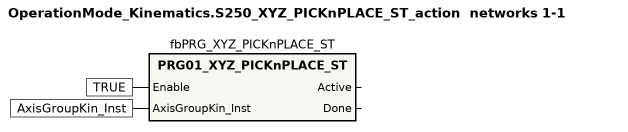
[picture p24: OperationMode_Kinematics.S250_XYZ_PICKnPLACE_ST_action (FBD) networks 1-1]
_FBD_ (* Function Block Diagram *)
NETWORK 1
	fbPRG_XYZ_PICKnPLACE_ST:PRG01_XYZ_PICKnPLACE_ST(Enable: TRUE, AxisGroupKin_Inst: AxisGroupKin_Inst)
_END_FBD_
(* the same logic as Structured Text *)
(* Network 1 *)
fbPRG_XYZ_PICKnPLACE_ST(Enable := TRUE, AxisGroupKin_Inst := AxisGroupKin_Inst);
END_ACTION

TRANSITION NOT referenced:
_FBD_ (* Function Block Diagram *)
NETWORK 1
	AND(AxisGroupKin_Inst.Out.General.Inverter.Connected[0], NOT AxisGroupKin_Inst.Out.General.Inverter.Referenced[0])
_END_FBD_
END_TRANSITION

TRANSITION referenced:
_FBD_ (* Function Block Diagram *)
NETWORK 1
	AND(AxisGroupKin_Inst.Out.General.Inverter.Connected[0], AxisGroupKin_Inst.Out.General.Inverter.Referenced[0])
_END_FBD_
END_TRANSITION

TRANSITION Homing done:
_FBD_ (* Function Block Diagram *)
NETWORK 1
	AND(AxisGroupKin_Inst.Out.General.Inverter.Connected[0], AxisGroupKin_Inst.Out.General.Inverter.Referenced[0])
_END_FBD_
END_TRANSITION

TRANSITION Automatic Mode:
_FBD_ (* Function Block Diagram *)
NETWORK 1
	AxisGroupKin_Inst.Out.General.Kin.Ready
_END_FBD_
(* the same logic as Structured Text *)
(* Network 1 *)
Automatic_Mode := AxisGroupKin_Inst.Out.General.Kin.Ready;
END_TRANSITION

TRANSITION Jog Mode:
_FBD_ (* Function Block Diagram *)
NETWORK 1
	NOT FALSE
_END_FBD_
(* the same logic as Structured Text *)
(* Network 1 *)
Jog_Mode := NOT FALSE;
END_TRANSITION

TRANSITION no Jog Mode:
_FBD_ (* Function Block Diagram *)
NETWORK 1
	FALSE
_END_FBD_
(* the same logic as Structured Text *)
(* Network 1 *)
no_Jog_Mode := FALSE;
END_TRANSITION

TRANSITION Start AND Enabled:
_FBD_ (* Function Block Diagram *)
NETWORK 1
	AND(TRUE, AxisGroupKin_Inst.Out.General.Kin.Ready)
_END_FBD_
END_TRANSITION

TRANSITION PRG1_Pick_and_Place_ST:
_FBD_ (* Function Block Diagram *)
NETWORK 1
	EQ(gKinExamples_Control[InstanceNumber].ProgramNumber, 1)
_END_FBD_
END_TRANSITION

TRANSITION Pick_and_Place_SFC:
_FBD_ (* Function Block Diagram *)
NETWORK 1
	EQ(gKinExamples_Control[InstanceNumber].ProgramNumber, 2)
_END_FBD_
END_TRANSITION

TRANSITION new Mode or Done:
_FBD_ (* Function Block Diagram *)
NETWORK 1
	OR(NE(gKinExamples_Control[InstanceNumber].ProgramNumber, 2), fbPRG_XYZ_PICKnPLACE_SFC.Done)
_END_FBD_
END_TRANSITION

TRANSITION XYZ_TARG_LIN_CIRC_ST:
_FBD_ (* Function Block Diagram *)
NETWORK 1
	EQ(gKinExamples_Control[InstanceNumber].ProgramNumber, 3)
_END_FBD_
END_TRANSITION

TRANSITION new Mode or Done:
_FBD_ (* Function Block Diagram *)
NETWORK 1
	OR(NE(gKinExamples_Control[InstanceNumber].ProgramNumber, 3), fbPRG_XYZ_TARG_LIN_CIRC_ST.Done)
_END_FBD_
END_TRANSITION

TRANSITION XYZ_TARG_LIN_CIRC_SFC:
_FBD_ (* Function Block Diagram *)
NETWORK 1
	EQ(gKinExamples_Control[InstanceNumber].ProgramNumber, 4)
_END_FBD_
END_TRANSITION

TRANSITION new Mode or Done:
_FBD_ (* Function Block Diagram *)
NETWORK 1
	OR(NE(gKinExamples_Control[InstanceNumber].ProgramNumber, 4), fbPRG_XYZ_TARG_LIN_CIRC_SFC.Done)
_END_FBD_
END_TRANSITION

TRANSITION XYZ_USER_ST:
_FBD_ (* Function Block Diagram *)
NETWORK 1
	EQ(gKinExamples_Control[InstanceNumber].ProgramNumber, 7)
_END_FBD_
END_TRANSITION

TRANSITION new Mode or Done:
_FBD_ (* Function Block Diagram *)
NETWORK 1
	OR(NE(gKinExamples_Control[InstanceNumber].ProgramNumber, 7), fbPRG_XYZ_USER_ST.Done)
_END_FBD_
END_TRANSITION

TRANSITION XYZ_USER_SFC:
_FBD_ (* Function Block Diagram *)
NETWORK 1
	EQ(gKinExamples_Control[InstanceNumber].ProgramNumber, 8)
_END_FBD_
END_TRANSITION

TRANSITION new Mode or Done:
_FBD_ (* Function Block Diagram *)
NETWORK 1
	OR(NE(gKinExamples_Control[InstanceNumber].ProgramNumber, 8), fbPRG_XYZ_USER_SFC.Done)
_END_FBD_
END_TRANSITION

TRANSITION FillQueue_LIN3D_with_Array_ST:
_FBD_ (* Function Block Diagram *)
NETWORK 1
	EQ(gKinExamples_Control[InstanceNumber].ProgramNumber, 5)
_END_FBD_
END_TRANSITION

TRANSITION new Mode or Done:
_FBD_ (* Function Block Diagram *)
NETWORK 1
	OR(NE(gKinExamples_Control[InstanceNumber].ProgramNumber, 5), fbPRG_XYZ_FillQueue_LIN3D_with_Array_ST.Done)
_END_FBD_
END_TRANSITION

TRANSITION FillQueue_LIN3D_with_Array_SFC:
_FBD_ (* Function Block Diagram *)
NETWORK 1
	EQ(gKinExamples_Control[InstanceNumber].ProgramNumber, 6)
_END_FBD_
END_TRANSITION

TRANSITION new Mode OR Done:
_FBD_ (* Function Block Diagram *)
NETWORK 1
	OR(NE(gKinExamples_Control[InstanceNumber].ProgramNumber, 6), fbPRG_XYZ_FillQueue_LIN3D_with_Array_SFC.Done)
_END_FBD_
END_TRANSITION

TRANSITION Jog Mode:
_FBD_ (* Function Block Diagram *)
NETWORK 1
	NOT FALSE
_END_FBD_
(* the same logic as Structured Text *)
(* Network 1 *)
Jog_Mode := NOT FALSE;
END_TRANSITION

TRANSITION new Mode or Done:
_FBD_ (* Function Block Diagram *)
NETWORK 1
	OR(NE(gKinExamples_Control[InstanceNumber].ProgramNumber, 1), fbPRG_XYZ_PICKnPLACE_ST.Done)
_END_FBD_
END_TRANSITION
END_FUNCTION_BLOCK

(* POU AxisGroupControl_Kinematics/Examples/PRG01_XYZ_PICKnPLACE_ST, ST *)
(*##############################################################################################################

	IMPORTANT NOTICE:
 	This example is a special and free service that demonstrates only the basic 
	approach to generating a PLC program as a non-binding sample. 
	SEW is not liable for the contents of the sample program.

	Name:			PRG_XYZ_PICKnPLACE_ST
	Job:			Example program		
					Sequence: XYZ_PICKnPLACE_P2 -> P3 -> P4 -> P3 -> P2 -> P1
					
################################################################################################################*)
FUNCTION_BLOCK  PRG01_XYZ_PICKnPLACE_ST
VAR_INPUT
	Enable : BOOL;
END_VAR
VAR_OUTPUT
	Active : BOOL;
	Done : BOOL;
END_VAR
VAR
	nState : INT := 0;
	fbRtrig : R_TRIG;
	i : INT;
END_VAR
VAR_IN_OUT
	AxisGroupKin_Inst											: ST_AxisGroupKin_Instance;
END_VAR
(* Initialisation at rising edge of VAR_INPUT Enable *)
fbRtrig(CLK:=Enable);
IF fbRtrig.Q THEN
	nState := 0;
	Active := TRUE;
END_IF

(* No execution, if Enable = False *)
IF (Enable = FALSE) THEN
	Done := FALSE;
	RETURN;
END_IF


CASE nState OF
0:	(*Start*)
	IF AxisGroupKin.ConfigDataAvailable THEN
		nState := 5;
	END_IF

5:	(* Up *)
	(* Initialize Kinematic Flags*)
	AxisGroupKin_Inst.In.Cp.Settings.PlusTargetCartABC:=FALSE;
	AxisGroupKin_Inst.In.Cp.Settings.UseMasterPosition:=FALSE;

(* TARGET_CART settings *)
	(* Motion Parameters *)
	AxisGroupKin_Inst.In.Target.Cart.Velocity := CART_VEL100;
	AxisGroupKin_Inst.In.Target.Cart.Acceleration := CART_ACC100;
	AxisGroupKin_Inst.In.Target.Cart.Deceleration := CART_DEC100;
	AxisGroupKin_Inst.In.Target.Cart.Jerk:=CART_Jerk100;
	AxisGroupKin_Inst.In.Target.Synchronization:= KIN_NO_SYNC;
	(* Coordinate System *)
	AxisGroupKin_Inst.In.Target.CoordSys:=KIN_KCS;

	AxisGroupKin_Inst.In.General.Mode := KIN_TARGET_CART;

	AxisGroupKin_Inst.In.Target.Position := XYZ_PICKnPLACE_P2;

	IF (MC_KinInProximity(Threshold := XYZ_PICKnPLACE_BlendingDistance,
			Position := AxisGroupKin_Inst.In.Target.Position,
			CoordSys := AxisGroupKin_Inst.In.Target.CoordSys,
			Dimension := 2#0000_0111, ActPos := AxisGroupKin_Inst.Out.General.Position)) THEN
		nState := 10;
	END_IF
	AxisGroupKin_Inst.In.Simu3D.Ctrl.Pen_TCP_WCS:=TRUE;

10:	(* Side *)
	AxisGroupKin_Inst.In.Target.Position := XYZ_PICKnPLACE_P3;
	IF (MC_KinInProximity(Threshold := XYZ_PICKnPLACE_BlendingDistance,
			Position := AxisGroupKin_Inst.In.Target.Position,
			CoordSys := AxisGroupKin_Inst.In.Target.CoordSys,
			Dimension := 2#0000_0111, ActPos := AxisGroupKin_Inst.Out.General.Position)) THEN
		nState := 20;
	END_IF

20:	(* Down *)
	AxisGroupKin_Inst.In.Target.Position := XYZ_PICKnPLACE_P4;
	IF (MC_KinInProximity(Threshold := 0.0,
			Position := AxisGroupKin_Inst.In.Target.Position,
			CoordSys := AxisGroupKin_Inst.In.Target.CoordSys,
			Dimension := 2#0000_0111, ActPos := AxisGroupKin_Inst.Out.General.Position)
			AND AxisGroupKin_Inst.Out.General.Standstill.ActCoordSys) THEN
		nState :=30;
	END_IF

30:	(* Up *)
	AxisGroupKin_Inst.In.Target.Position := XYZ_PICKnPLACE_P3;
	IF (MC_KinInProximity(Threshold := XYZ_PICKnPLACE_BlendingDistance,
			Position := AxisGroupKin_Inst.In.Target.Position,
			CoordSys := AxisGroupKin_Inst.In.Target.CoordSys,
			Dimension := 2#0000_0111, ActPos := AxisGroupKin_Inst.Out.General.Position)) THEN
		nState := 40;
	END_IF

40:	(* Side *)
	AxisGroupKin_Inst.In.Target.Position := XYZ_PICKnPLACE_P2;
	IF (MC_KinInProximity(Threshold := XYZ_PICKnPLACE_BlendingDistance,
			Position := AxisGroupKin_Inst.In.Target.Position,
			CoordSys := AxisGroupKin_Inst.In.Target.CoordSys,
			Dimension := 2#0000_0111, ActPos := AxisGroupKin_Inst.Out.General.Position)) THEN
		nState := 50;
	END_IF

50:	(* Down *)
	AxisGroupKin_Inst.In.Target.Position := XYZ_PICKnPLACE_P1;
	IF (MC_KinInProximity(Threshold := 0.0,
			Position := AxisGroupKin_Inst.In.Target.Position,
			CoordSys := AxisGroupKin_Inst.In.Target.CoordSys,
			Dimension := 2#0000_0111, ActPos := AxisGroupKin_Inst.Out.General.Position)
			AND AxisGroupKin_Inst.Out.General.Standstill.ActCoordSys) THEN
		AxisGroupKin_Inst.In.Simu3D.Ctrl.Pen_TCP_WCS:=FALSE;
		Done := TRUE;
		Active := FALSE;
	END_IF

ELSE
;

END_CASE
END_FUNCTION_BLOCK

(* POU AxisGroupControl_Kinematics/Examples/PRG02_XYZ_PICKnPLACE_SFC, SFC *)
(*##############################################################################################################

	IMPORTANT NOTICE:
 	This example is a special and free service that demonstrates only the basic 
	approach to generating a PLC program as a non-binding sample. 
	SEW is not liable for the contents of the sample program.

	Name:			PRG_XYZ_PICKnPLACE_SFC
	Job:			Example program		
					Sequence: XYZ_PICKnPLACE_P2 -> P3 -> P4 -> P3 -> P2 -> P1	

################################################################################################################*)
FUNCTION_BLOCK PRG02_XYZ_PICKnPLACE_SFC
VAR_INPUT
	SFCReset:BOOL;
	(*SFCInit:BOOL;*)
	SFCPause:BOOL;

	SFCTipMode:BOOL;
	SFCTip:BOOL;
	SFCEnableLimit:BOOL;
	SFCQuitError:BOOL;
END_VAR
VAR_OUTPUT
	SFCTrans:BOOL;
	SFCError:BOOL;
	SFCErrorStep:STRING;
	SFCErrorPOU:STRING;
	SFCCurrentStep:STRING;
	Done:BOOL;
END_VAR
VAR

END_VAR
VAR_IN_OUT
	AxisGroupKin_Inst											: ST_AxisGroupKin_Instance;
END_VAR
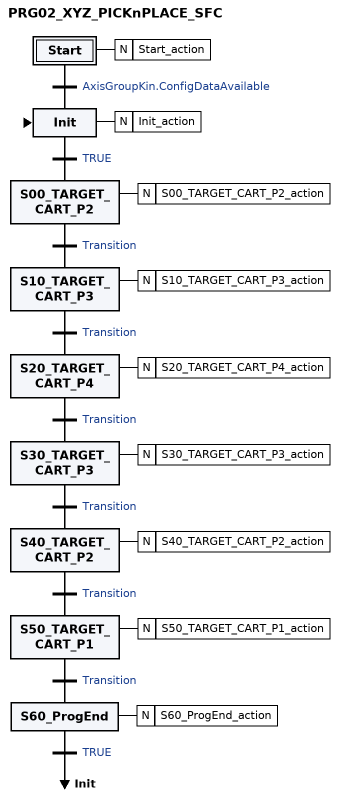
INITIAL_STEP Start:
	Start_action(N);
END_STEP
TRANSITION FROM Start TO Init := AxisGroupKin.ConfigDataAvailable;
END_TRANSITION
STEP Init:
	Init_action(N);
END_STEP
TRANSITION FROM Init TO S00_TARGET_CART_P2 := TRUE;
END_TRANSITION
STEP S00_TARGET_CART_P2:
	S00_TARGET_CART_P2_action(N);
END_STEP
TRANSITION FROM S00_TARGET_CART_P2 TO S10_TARGET_CART_P3 := Transition;
END_TRANSITION
STEP S10_TARGET_CART_P3:
	S10_TARGET_CART_P3_action(N);
END_STEP
TRANSITION FROM S10_TARGET_CART_P3 TO S20_TARGET_CART_P4 := Transition;
END_TRANSITION
STEP S20_TARGET_CART_P4:
	S20_TARGET_CART_P4_action(N);
END_STEP
TRANSITION FROM S20_TARGET_CART_P4 TO S30_TARGET_CART_P3 := Transition;
END_TRANSITION
STEP S30_TARGET_CART_P3:
	S30_TARGET_CART_P3_action(N);
END_STEP
TRANSITION FROM S30_TARGET_CART_P3 TO S40_TARGET_CART_P2 := Transition;
END_TRANSITION
STEP S40_TARGET_CART_P2:
	S40_TARGET_CART_P2_action(N);
END_STEP
TRANSITION FROM S40_TARGET_CART_P2 TO S50_TARGET_CART_P1 := Transition;
END_TRANSITION
STEP S50_TARGET_CART_P1:
	S50_TARGET_CART_P1_action(N);
END_STEP
TRANSITION FROM S50_TARGET_CART_P1 TO S60_ProgEnd := Transition;
END_TRANSITION
STEP S60_ProgEnd:
	S60_ProgEnd_action(N);
END_STEP
TRANSITION FROM S60_ProgEnd TO Init := TRUE;
END_TRANSITION

ACTION Start_action:
Done:=FALSE;
END_ACTION

ACTION Init_action:
(* Initialize Kinematic Flags*)
	AxisGroupKin_Inst.In.Cp.Settings.PlusTargetCartABC:=FALSE;
	AxisGroupKin_Inst.In.Cp.Settings.UseMasterPosition:=FALSE;

(* TARGET_CART settings *)
	(* Motion Parameters *)
	AxisGroupKin_Inst.In.Target.Cart.Velocity := CART_VEL100;
	AxisGroupKin_Inst.In.Target.Cart.Acceleration := CART_ACC100;
	AxisGroupKin_Inst.In.Target.Cart.Deceleration := CART_DEC100;
	AxisGroupKin_Inst.In.Target.Cart.Jerk := CART_Jerk100;
	AxisGroupKin_Inst.In.Target.Synchronization := KIN_NO_SYNC;
	(* Coordinate System *)
	AxisGroupKin_Inst.In.Target.CoordSys := KIN_KCS;

	AxisGroupKin_Inst.In.General.Mode := KIN_TARGET_CART;
END_ACTION

ACTION S00_TARGET_CART_P2_action:
AxisGroupKin_Inst.In.Target.Position := XYZ_PICKnPLACE_P2;
END_ACTION

ACTION S10_TARGET_CART_P3_action:
AxisGroupKin_Inst.In.Target.Position := XYZ_PICKnPLACE_P3;
END_ACTION

ACTION S20_TARGET_CART_P4_action:
AxisGroupKin_Inst.In.Target.Position := XYZ_PICKnPLACE_P4;
END_ACTION

ACTION S30_TARGET_CART_P3_action:
AxisGroupKin_Inst.In.Target.Position := XYZ_PICKnPLACE_P3;
END_ACTION

ACTION S40_TARGET_CART_P2_action:
AxisGroupKin_Inst.In.Target.Position := XYZ_PICKnPLACE_P2;
END_ACTION

ACTION S50_TARGET_CART_P1_action:
AxisGroupKin_Inst.In.Target.Position := XYZ_PICKnPLACE_P1;
END_ACTION

ACTION S60_ProgEnd_action:
Done:=TRUE;
END_ACTION

TRANSITION Transition:
MC_KinInProximity(Threshold := XYZ_PICKnPLACE_BlendingDistance,
			Position := AxisGroupKin_Inst.In.Target.Position,
			CoordSys := AxisGroupKin_Inst.In.Target.CoordSys,
			Dimension := 2#0000_0111, ActPos := AxisGroupKin_Inst.Out.General.Position)
END_TRANSITION

TRANSITION Transition:
MC_KinInProximity(Threshold := XYZ_PICKnPLACE_BlendingDistance,
			Position := AxisGroupKin_Inst.In.Target.Position,
			CoordSys := AxisGroupKin_Inst.In.Target.CoordSys,
			Dimension := 2#0000_0111, ActPos := AxisGroupKin_Inst.Out.General.Position)
END_TRANSITION

TRANSITION Transition:
MC_KinInProximity(Threshold := 0.0,
			Position := AxisGroupKin_Inst.In.Target.Position,
			CoordSys := AxisGroupKin_Inst.In.Target.CoordSys,
			Dimension := 2#0000_0111, ActPos := AxisGroupKin_Inst.Out.General.Position)
AND
AxisGroupKin_Inst.Out.General.Standstill.ActCoordSys
END_TRANSITION

TRANSITION Transition:
MC_KinInProximity(Threshold := XYZ_PICKnPLACE_BlendingDistance,
			Position := AxisGroupKin_Inst.In.Target.Position,
			CoordSys := AxisGroupKin_Inst.In.Target.CoordSys,
			Dimension := 2#0000_0111, ActPos := AxisGroupKin_Inst.Out.General.Position)
END_TRANSITION

TRANSITION Transition:
MC_KinInProximity(Threshold := XYZ_PICKnPLACE_BlendingDistance,
			Position := AxisGroupKin_Inst.In.Target.Position,
			CoordSys := AxisGroupKin_Inst.In.Target.CoordSys,
			Dimension := 2#0000_0111, ActPos := AxisGroupKin_Inst.Out.General.Position)
END_TRANSITION

TRANSITION Transition:
MC_KinInProximity(Threshold := 0.0,
			Position := AxisGroupKin_Inst.In.Target.Position,
			CoordSys := AxisGroupKin_Inst.In.Target.CoordSys,
			Dimension := 2#0000_0111, ActPos := AxisGroupKin_Inst.Out.General.Position)
AND
AxisGroupKin_Inst.Out.General.Standstill.ActCoordSys
END_TRANSITION
END_FUNCTION_BLOCK

(* POU AxisGroupControl_Kinematics/Examples/PRG03_XYZ_TARG_LIN_CIRC_ST, ST *)
(*##############################################################################################################

	IMPORTANT NOTICE:
 	This example is a special and free service that demonstrates only the basic 
	approach to generating a PLC program as a non-binding sample. 
	SEW is not liable for the contents of the sample program.

	Name:			PRG_XYZ_TARG_LIN_CIRC_ST
	Job:			Example program			
					Sequence: TARGET_CART to XYZ_TARG_LIN_CIRC_P1 -> LIN_XY to P2 -> CIRC_XZ with R3/A3 -> LIN_3D to P4 -> LIN_XY to P1

################################################################################################################*)
FUNCTION_BLOCK PRG03_XYZ_TARG_LIN_CIRC_ST
VAR_INPUT
	Enable : BOOL;
END_VAR
VAR_OUTPUT
	Active : BOOL;
	Done : BOOL;
END_VAR
VAR
	nState : INT;
	fbRtrig : R_TRIG;
END_VAR
VAR_IN_OUT
	AxisGroupKin_Inst											: ST_AxisGroupKin_Instance;
END_VAR
(* Initialisation at rising edge of VAR_INPUT Enable *)
fbRtrig(CLK:=Enable);
IF fbRtrig.Q THEN
	nState	:= 0;
	Active := TRUE;
END_IF

(* No execution, if Enable = False *)
IF NOT Enable THEN
	Done := FALSE;
	RETURN;
END_IF


CASE nState OF
0:	(*Start*)
	IF AxisGroupKin.ConfigDataAvailable THEN
		nState := 5;
	END_IF
5:	(* TARGET_CART to XYZ_TARG_LIN_CIRC_P1 *)
	(* Initialize Kinematic Flags*)
	AxisGroupKin_Inst.In.Cp.Settings.PlusTargetCartABC:=FALSE;
	AxisGroupKin_Inst.In.Cp.Settings.UseMasterPosition:=FALSE;

(* TARGET_CART settings *)
	(* Motion Parameters *)
	AxisGroupKin_Inst.In.Target.Cart.Acceleration := CART_ACC50;
	AxisGroupKin_Inst.In.Target.Cart.Deceleration := CART_DEC50;
	AxisGroupKin_Inst.In.Target.Cart.Velocity := CART_VEL50;
	AxisGroupKin_Inst.In.Target.Cart.Jerk:=CART_Jerk100;
	AxisGroupKin_Inst.In.Target.Synchronization:= KIN_NO_SYNC;
	(* Coordinate System *)
	AxisGroupKin_Inst.In.Target.CoordSys:=KIN_KCS;

	AxisGroupKin_Inst.In.General.Mode := KIN_TARGET_CART;

	AxisGroupKin_Inst.In.Target.Position := XYZ_TARG_LIN_CIRC_P1;
	IF (MC_KinInProximity(Threshold := 0.0,
			Position := AxisGroupKin_Inst.In.Target.Position,
			CoordSys := AxisGroupKin_Inst.In.Target.CoordSys,
			Dimension := 2#0000_0111, ActPos := AxisGroupKin_Inst.Out.General.Position)
			AND AxisGroupKin_Inst.Out.General.Standstill.ActCoordSys) THEN
		nState := 10;
	END_IF

10:	(* Straight line to XYZ_TARG_LIN_CIRC_P2, as soon as XYZ_TARG_LIN_CIRC_P1 has been reached *)

		AxisGroupKin_Inst.In.General.Mode := KIN_LIN_XY;
		AxisGroupKin_Inst.In.Cp.Segment.Position := XYZ_TARG_LIN_CIRC_P2;
(* CP motion parameters *)
		(* settings for whole path / all segments *)
		AxisGroupKin_Inst.In.Cp.Path.VelocityPercentage:=100;
		AxisGroupKin_Inst.In.Cp.Path.FidelityPercentage :=100;
		(* Settings for the segment, which should be added to the queue *)
		AxisGroupKin_Inst.In.Cp.Segment.Translation.Velocity := 1000;
		AxisGroupKin_Inst.In.Cp.Segment.Translation.Acceleration := 100;
		AxisGroupKin_Inst.In.Cp.Segment.Translation.Deceleration := 100;
		AxisGroupKin_Inst.In.Cp.Segment.Translation.Jerk := 100;
		AxisGroupKin_Inst.In.Cp.Segment.Blending.Distance := 50;
		AxisGroupKin_Inst.In.Cp.Segment.Blending.LimitationPercentage := 50;

		AxisGroupKin_Inst.In.Cp.Segment.ID := AxisGroupKin_Inst.In.Cp.Segment.ID + 1;	(* Change the SegmentID to add the segment to the queue *)

		AxisGroupKin_Inst.In.Simu3D.Ctrl.Pen_TCP_WCS := TRUE;

		nState := 20;

20:	(* A circle section is written into the queue directly after the straight line *)
	IF (AxisGroupKin_Inst.Out.Cp.Queue.LastMappedSegID = AxisGroupKin_Inst.In.Cp.Segment.ID) THEN (* Wait until the segment was added to the queue; this is not required if FB_KinControl is executed in the same task *)
		AxisGroupKin_Inst.In.General.Mode := KIN_CIRC_ZX;
		(* Parameters to define the circle *)
		AxisGroupKin_Inst.In.Cp.Segment.Circ.Mode := KIN_RADIUS_ANGLE;	(* Define the circle with the radius and angle *)
		AxisGroupKin_Inst.In.Cp.Segment.Circ.Direction := KIN_CW;	(* Draw circle ClockWise *)
		AxisGroupKin_Inst.In.Cp.Segment.Circ.Radius := XYZ_TARG_LIN_CIRC_R3;
		AxisGroupKin_Inst.In.Cp.Segment.Circ.Angle := XYZ_TARG_LIN_CIRC_A3;


		AxisGroupKin_Inst.In.Cp.Segment.ID := AxisGroupKin_Inst.In.Cp.Segment.ID + 1;
		nState := 30;
	END_IF

30:	(* A Straight line to XYZ_TARG_LIN_CIRC_P4 is written into the queue directly after the circle section
		-> Blending to the straight line is performed automatically *)
	IF (AxisGroupKin_Inst.Out.Cp.Queue.LastMappedSegID = AxisGroupKin_Inst.In.Cp.Segment.ID) THEN
		AxisGroupKin_Inst.In.General.Mode := KIN_LIN_3D;
		AxisGroupKin_Inst.In.Cp.Segment.Position := XYZ_TARG_LIN_CIRC_P4;


		AxisGroupKin_Inst.In.Cp.Segment.ID := AxisGroupKin_Inst.In.Cp.Segment.ID + 1;
		nState := 40;
	END_IF

40:	(* Straight line to XYZ_TARG_LIN_CIRC_P1 is written into the queue directly after the previous straight line
		-> Blending to the straight line is performed automatically *)
	IF (AxisGroupKin_Inst.Out.Cp.Queue.LastMappedSegID = AxisGroupKin_Inst.In.Cp.Segment.ID) THEN
		AxisGroupKin_Inst.In.General.Mode := KIN_LIN_XY;
		AxisGroupKin_Inst.In.Cp.Segment.Position := XYZ_TARG_LIN_CIRC_P1;


		AxisGroupKin_Inst.In.Cp.Segment.ID := AxisGroupKin_Inst.In.Cp.Segment.ID + 1;
		nState := 50;
	END_IF

50:	(* Program end, as soon as XYZ_TARG_LIN_CIRC_P1 has been reached *)
	IF (AxisGroupKin_Inst.Out.Cp.Path.EndReached)
	AND (AxisGroupKin_Inst.Out.Cp.Queue.LastMappedSegID = AxisGroupKin_Inst.In.Cp.Segment.ID) THEN
		Done := TRUE;
		Active := FALSE;
		AxisGroupKin_Inst.In.Simu3D.Ctrl.Pen_TCP_WCS := FALSE;
	END_IF

ELSE
;

END_CASE
END_FUNCTION_BLOCK

(* POU AxisGroupControl_Kinematics/Examples/PRG04_XYZ_TARG_LIN_CIRC_SFC, SFC *)
(*##############################################################################################################

	IMPORTANT NOTICE:
 	This example is a special and free service that demonstrates only the basic 
	approach to generating a PLC program as a non-binding sample. 
	SEW is not liable for the contents of the sample program.

	Name:			PRG_XYZ_TARG_LIN_CIRC_SFC
	Job:			Example program			
					Sequence: TARGET_CART to XYZ_TARG_LIN_CIRC_P1 -> LIN_XY to P2 -> CIRC_XZ with R3/A3 -> LIN_3D to P4 -> LIN_XY to P1

################################################################################################################*)
FUNCTION_BLOCK PRG04_XYZ_TARG_LIN_CIRC_SFC
VAR_INPUT
	SFCReset:BOOL;
	(*SFCInit:BOOL;*)
	SFCPause:BOOL;

	SFCTipMode:BOOL;
	SFCTip:BOOL;
	SFCEnableLimit:BOOL;
	SFCQuitError:BOOL;

END_VAR
VAR_OUTPUT
	SFCTrans:BOOL;
	SFCError:BOOL;
	SFCErrorStep:STRING;
	SFCErrorPOU:STRING;
(*	SFCErrorAnalyzation:STRING;*)
	SFCCurrentStep:STRING;
	Done:BOOL;
END_VAR
VAR

END_VAR
VAR_IN_OUT
	AxisGroupKin_Inst											: ST_AxisGroupKin_Instance;
END_VAR
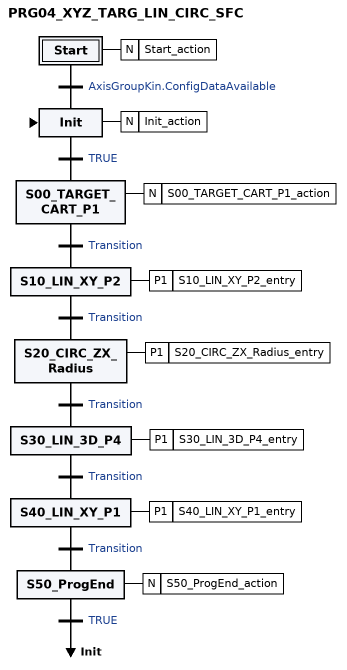
INITIAL_STEP Start:
	Start_action(N);
END_STEP
TRANSITION FROM Start TO Init := AxisGroupKin.ConfigDataAvailable;
END_TRANSITION
STEP Init:
	Init_action(N);
END_STEP
TRANSITION FROM Init TO S00_TARGET_CART_P1 := TRUE;
END_TRANSITION
STEP S00_TARGET_CART_P1:
	S00_TARGET_CART_P1_action(N);
END_STEP
TRANSITION FROM S00_TARGET_CART_P1 TO S10_LIN_XY_P2 := Transition;
END_TRANSITION
STEP S10_LIN_XY_P2:
	S10_LIN_XY_P2_entry(P1);
END_STEP
TRANSITION FROM S10_LIN_XY_P2 TO S20_CIRC_ZX_Radius := Transition;
END_TRANSITION
STEP S20_CIRC_ZX_Radius:
	S20_CIRC_ZX_Radius_entry(P1);
END_STEP
TRANSITION FROM S20_CIRC_ZX_Radius TO S30_LIN_3D_P4 := Transition;
END_TRANSITION
STEP S30_LIN_3D_P4:
	S30_LIN_3D_P4_entry(P1);
END_STEP
TRANSITION FROM S30_LIN_3D_P4 TO S40_LIN_XY_P1 := Transition;
END_TRANSITION
STEP S40_LIN_XY_P1:
	S40_LIN_XY_P1_entry(P1);
END_STEP
TRANSITION FROM S40_LIN_XY_P1 TO S50_ProgEnd := Transition;
END_TRANSITION
STEP S50_ProgEnd:
	S50_ProgEnd_action(N);
END_STEP
TRANSITION FROM S50_ProgEnd TO Init := TRUE;
END_TRANSITION

ACTION Start_action:
Done:=FALSE;
END_ACTION

ACTION Init_action:
(* Initialize Kinematic Flags*)
	AxisGroupKin_Inst.In.Cp.Settings.PlusTargetCartABC:=FALSE;
	AxisGroupKin_Inst.In.Cp.Settings.UseMasterPosition:=FALSE;

(* TARGET_CART settings *)
	(* Motion Parameters *)
	AxisGroupKin_Inst.In.Target.Cart.Acceleration := CART_ACC50;
	AxisGroupKin_Inst.In.Target.Cart.Deceleration := CART_DEC50;
	AxisGroupKin_Inst.In.Target.Cart.Velocity := CART_VEL50;
	AxisGroupKin_Inst.In.Target.Cart.Jerk:=CART_Jerk100;
	AxisGroupKin_Inst.In.Target.Synchronization:= KIN_NO_SYNC;
	(* Coordinate System *)
	AxisGroupKin_Inst.In.Target.CoordSys:=KIN_KCS;

	AxisGroupKin_Inst.In.General.Mode := KIN_TARGET_CART;
END_ACTION

ACTION S00_TARGET_CART_P1_action:
AxisGroupKin_Inst.In.Target.Position :=  XYZ_TARG_LIN_CIRC_P1;
END_ACTION

ACTION S10_LIN_XY_P2_entry:
(* Straight line to XYZ_TARG_LIN_CIRC_P2, as soon as XYZ_TARG_LIN_CIRC_P1 has been reached *)

		AxisGroupKin_Inst.In.General.Mode := KIN_LIN_XY;
		AxisGroupKin_Inst.In.Cp.Segment.Position := XYZ_TARG_LIN_CIRC_P2;
(* CP motion parameters *)
		(* settings for whole path / all segments *)
		AxisGroupKin_Inst.In.Cp.Path.VelocityPercentage:=100;
		AxisGroupKin_Inst.In.Cp.Path.FidelityPercentage :=100;
		(* Settings for the segment, which should be added to the queue *)
		AxisGroupKin_Inst.In.Cp.Segment.Translation.Velocity := 1000;
		AxisGroupKin_Inst.In.Cp.Segment.Translation.Acceleration := 100;
		AxisGroupKin_Inst.In.Cp.Segment.Translation.Deceleration := 100;
		AxisGroupKin_Inst.In.Cp.Segment.Translation.Jerk := 100;
		AxisGroupKin_Inst.In.Cp.Segment.Blending.Distance := 50;
		AxisGroupKin_Inst.In.Cp.Segment.Blending.LimitationPercentage := 50;

		AxisGroupKin_Inst.In.Cp.Segment.ID := AxisGroupKin_Inst.In.Cp.Segment.ID + 1;	(* Change the SegmentID to add the segment to the queue *)

		AxisGroupKin_Inst.In.Simu3D.Ctrl.Pen_TCP_WCS := TRUE;
END_ACTION

ACTION S20_CIRC_ZX_Radius_entry:
AxisGroupKin_Inst.In.General.Mode := KIN_CIRC_ZX;
(* Parameters to define the circle *)
AxisGroupKin_Inst.In.Cp.Segment.Circ.Mode := KIN_RADIUS_ANGLE;	(* Define the circle with the radius and angle *)
AxisGroupKin_Inst.In.Cp.Segment.Circ.Direction := KIN_CW;	(* Draw circle ClockWise *)
AxisGroupKin_Inst.In.Cp.Segment.Circ.Radius := XYZ_TARG_LIN_CIRC_R3;
AxisGroupKin_Inst.In.Cp.Segment.Circ.Angle := XYZ_TARG_LIN_CIRC_A3;


AxisGroupKin_Inst.In.Cp.Segment.ID := AxisGroupKin_Inst.In.Cp.Segment.ID + 1;
END_ACTION

ACTION S30_LIN_3D_P4_entry:
AxisGroupKin_Inst.In.General.Mode := KIN_LIN_3D;
AxisGroupKin_Inst.In.Cp.Segment.Position := XYZ_TARG_LIN_CIRC_P4;


AxisGroupKin_Inst.In.Cp.Segment.ID := AxisGroupKin_Inst.In.Cp.Segment.ID + 1;
END_ACTION

ACTION S40_LIN_XY_P1_entry:
AxisGroupKin_Inst.In.General.Mode := KIN_LIN_XY;
AxisGroupKin_Inst.In.Cp.Segment.Position := XYZ_TARG_LIN_CIRC_P1;


AxisGroupKin_Inst.In.Cp.Segment.ID := AxisGroupKin_Inst.In.Cp.Segment.ID + 1;
END_ACTION

ACTION S50_ProgEnd_action:
Done := TRUE;
AxisGroupKin_Inst.In.Simu3D.Ctrl.Pen_TCP_WCS := FALSE;  (* Process Off *)
END_ACTION

TRANSITION Transition:
MC_KinInProximity(Threshold := 0.0,
			Position := AxisGroupKin_Inst.In.Target.Position,
			CoordSys := AxisGroupKin_Inst.In.Target.CoordSys,
			Dimension := 2#0000_0111, ActPos := AxisGroupKin_Inst.Out.General.Position)
AND
AxisGroupKin_Inst.Out.General.Standstill.ActCoordSys
END_TRANSITION

TRANSITION Transition:
(* Wait until the segment was added to the queue; this is not required if FB_KinControl is executed in the same task *)
AxisGroupKin_Inst.Out.Cp.Queue.LastMappedSegID = AxisGroupKin_Inst.In.Cp.Segment.ID
END_TRANSITION

TRANSITION Transition:
(* Wait until the segment was added to the queue; this is not required if FB_KinControl is executed in the same task *)
AxisGroupKin_Inst.Out.Cp.Queue.LastMappedSegID = AxisGroupKin_Inst.In.Cp.Segment.ID
END_TRANSITION

TRANSITION Transition:
(* Wait until the segment was added to the queue; this is not required if FB_KinControl is executed in the same task *)
AxisGroupKin_Inst.Out.Cp.Queue.LastMappedSegID = AxisGroupKin_Inst.In.Cp.Segment.ID
END_TRANSITION

TRANSITION Transition:
(AxisGroupKin_Inst.Out.Cp.Path.EndReached) AND
(AxisGroupKin_Inst.Out.Cp.Queue.LastMappedSegID = AxisGroupKin_Inst.In.Cp.Segment.ID)
END_TRANSITION
END_FUNCTION_BLOCK

(* POU AxisGroupControl_Kinematics/Examples/PRG05_XYZ_FillQueue_LIN3D_with_Array_ST, ST *)
(*##############################################################################################################

	IMPORTANT NOTICE:
 	This example is a special and free service that demonstrates only the basic 
	approach to generating a PLC program as a non-binding sample. 
	SEW is not liable for the contents of the sample program.

	Name:			PRG_XYZ_FillQueue_LIN3D_with_Array_ST
	Job:			Example program			

################################################################################################################*)
FUNCTION_BLOCK PRG05_XYZ_FillQueue_LIN3D_with_Array_ST

VAR_INPUT
	Enable: BOOL;
END_VAR
VAR_OUTPUT
	Active: BOOL;
	Done: BOOL;
END_VAR
VAR
	nState : INT := 0;
	i:INT:=1;
END_VAR
VAR_IN_OUT
	AxisGroupKin_Inst											: ST_AxisGroupKin_Instance;
END_VAR
IF NOT Enable THEN
	Done:=FALSE;
	Active := FALSE;
	i:=1;
	nState:=0;
	RETURN;
END_IF
CASE nState OF
0:	(*Start*)
	IF AxisGroupKin.ConfigDataAvailable THEN
		nState := 5;
	END_IF

5:	(* Initialization and TARGET_CART to last point in queue *)

	(* Initialize kinematics flags*)
	AxisGroupKin_Inst.In.Cp.Settings.PlusTargetCartABC :=FALSE;
	AxisGroupKin_Inst.In.Cp.Settings.UseMasterPosition:=FALSE;

(* CP settings *)
	(* Initialize SegID *)
	AxisGroupKin_Inst.In.Cp.Segment.ID := AxisGroupKin_Inst.Out.Cp.Queue.LastMappedSegID;
	(* Initialize global point array *)
	points[1].x:=10;	points[1].y:=100;	points[1].z:=50;
	points[2].x:=10;	points[2].y:=200;	points[2].z:=100;
	points[3].x:=50;	points[3].y:=300;	points[3].z:=50;
	points[4].x:=100;	points[4].y:=350;	points[4].z:=100;
	points[5].x:=200;	points[5].y:=300;	points[5].z:=50;
	points[6].x:=300;	points[6].y:=200;	points[6].z:=100;
	points[7].x:=300;	points[7].y:=100;	points[7].z:=50;
	points[8].x:=200;	points[8].y:=50;	points[8].z:=100;
	points[9].x:=100;	points[9].y:=10;	points[9].z:=50;
	points[10].x:=50;	points[10].y:=50;	points[10].z:=100;
	(* motion parameters for CP modes *)
	AxisGroupKin_Inst.In.Cp.Segment.Translation.Velocity := 100;
	AxisGroupKin_Inst.In.Cp.Segment.Translation.Acceleration := 100;
	AxisGroupKin_Inst.In.Cp.Segment.Translation.Deceleration := 100;
	AxisGroupKin_Inst.In.Cp.Segment.Translation.Jerk := 100;
	AxisGroupKin_Inst.In.Cp.Segment.Blending.Distance := 30;
	AxisGroupKin_Inst.In.Cp.Segment.Blending.LimitationPercentage := 50;
	AxisGroupKin_Inst.In.Cp.Segment.Mode := KIN_CONTINUOUS_PATH;
	AxisGroupKin_Inst.In.Cp.Path.VelocityPercentage:=100;
	AxisGroupKin_Inst.In.Cp.Path.FidelityPercentage :=100;

(* TARGET_CART settings *)
	(* Set motion parameters for target mode*)
	AxisGroupKin_Inst.In.Target.Cart.Acceleration := CART_ACC50;
	AxisGroupKin_Inst.In.Target.Cart.Deceleration := CART_DEC50;
	AxisGroupKin_Inst.In.Target.Cart.Velocity := CART_VEL50;
	AxisGroupKin_Inst.In.Target.Cart.Jerk:=CART_Jerk100;
	AxisGroupKin_Inst.In.Target.CoordSys := KIN_KCS;
	AxisGroupKin_Inst.In.Target.Synchronization:= KIN_NO_SYNC;
	(* move to last point in array *)
	AxisGroupKin_Inst.In.Target.Position[1] := points[10].x;
	AxisGroupKin_Inst.In.Target.Position[2] := points[10].y;
	AxisGroupKin_Inst.In.Target.Position[3] := points[10].z;

	AxisGroupKin_Inst.In.General.Mode := KIN_TARGET_CART;

	IF (MC_KinInProximity(Threshold := 0.0,
			Position := AxisGroupKin_Inst.In.Target.Position,
			CoordSys := AxisGroupKin_Inst.In.Target.CoordSys,
			Dimension := 2#0000_0111, ActPos := AxisGroupKin_Inst.Out.General.Position)
			AND AxisGroupKin_Inst.Out.General.Standstill.ActCoordSys) THEN
		nState := 10;
	END_IF
10:	(*Fill Queue *)
	IF i <=10 THEN
		AxisGroupKin_Inst.In.Simu3D.Ctrl.Pen_TCP_WCS :=TRUE;
		IF AxisGroupKin_Inst.Out.Cp.Queue.LastMappedSegID = AxisGroupKin_Inst.In.Cp.Segment.ID THEN
			AxisGroupKin_Inst.In.General.Mode := KIN_LIN_3D;
			AxisGroupKin_Inst.In.Cp.Segment.Position[1] := points[i].x;
			AxisGroupKin_Inst.In.Cp.Segment.Position[2] := points[i].y;
			AxisGroupKin_Inst.In.Cp.Segment.Position[3] := points[i].z;
			AxisGroupKin_Inst.In.Cp.Segment.ID := AxisGroupKin_Inst.In.Cp.Segment.ID + 1;
			i:=i+1;
		END_IF
	ELSIF AxisGroupKin_Inst.Out.Cp.Path.EndReached THEN
		Done := TRUE;
		Active := FALSE;
		AxisGroupKin_Inst.In.Simu3D.Ctrl.Pen_TCP_WCS := FALSE;
	END_IF
END_CASE
END_FUNCTION_BLOCK

(* POU AxisGroupControl_Kinematics/Examples/PRG06_XYZ_FillQueue_LIN3D_with_Array_SFC, SFC *)
(*##############################################################################################################

	IMPORTANT NOTICE:
 	This example is a special and free service that demonstrates only the basic 
	approach to generating a PLC program as a non-binding sample. 
	SEW is not liable for the contents of the sample program.

	Name:			PRG_XYZ_FillQueue_LIN3D_with_Array_SFC
	Job:			Example program		

################################################################################################################*)
FUNCTION_BLOCK PRG06_XYZ_FillQueue_LIN3D_with_Array_SFC
VAR_INPUT
	SFCReset:BOOL;
	(*SFCInit:BOOL;*)
	SFCPause:BOOL;

	SFCTipMode:BOOL;
	SFCTip:BOOL;
	SFCEnableLimit:BOOL;
	SFCQuitError:BOOL;

END_VAR
VAR_OUTPUT
	SFCTrans:BOOL;
	SFCError:BOOL;
	SFCErrorStep:STRING;
	SFCErrorPOU:STRING;
	SFCCurrentStep:STRING;
	Done:BOOL;
END_VAR
VAR
	i:INT;
END_VAR
VAR_IN_OUT
	AxisGroupKin_Inst	: ST_AxisGroupKin_Instance;
END_VAR
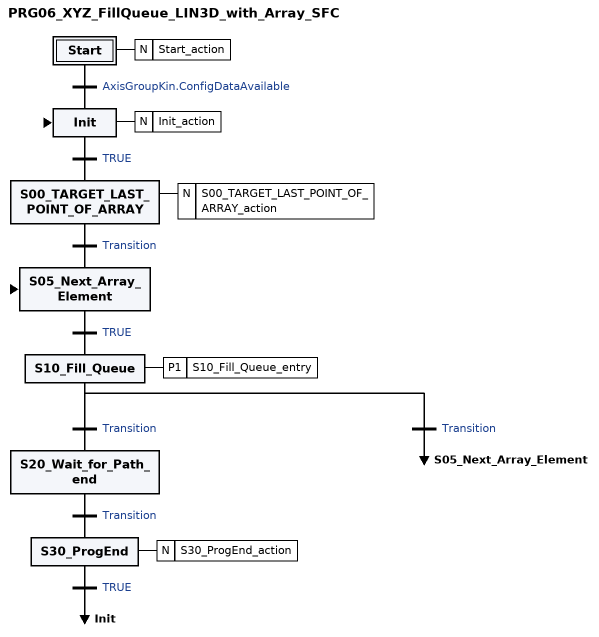
INITIAL_STEP Start:
	Start_action(N);
END_STEP
TRANSITION FROM Start TO Init := AxisGroupKin.ConfigDataAvailable;
END_TRANSITION
STEP Init:
	Init_action(N);
END_STEP
TRANSITION FROM Init TO S00_TARGET_LAST_POINT_OF_ARRAY := TRUE;
END_TRANSITION
STEP S00_TARGET_LAST_POINT_OF_ARRAY:
	S00_TARGET_LAST_POINT_OF_ARRAY_action(N);
END_STEP
TRANSITION FROM S00_TARGET_LAST_POINT_OF_ARRAY TO S05_Next_Array_Element := Transition;
END_TRANSITION
STEP S05_Next_Array_Element:
END_STEP
TRANSITION FROM S05_Next_Array_Element TO S10_Fill_Queue := TRUE;
END_TRANSITION
STEP S10_Fill_Queue:
	S10_Fill_Queue_entry(P1);
END_STEP
TRANSITION FROM S10_Fill_Queue TO S20_Wait_for_Path_end := Transition;
END_TRANSITION
TRANSITION FROM S10_Fill_Queue TO S05_Next_Array_Element := Transition;
END_TRANSITION
STEP S20_Wait_for_Path_end:
END_STEP
TRANSITION FROM S20_Wait_for_Path_end TO S30_ProgEnd := Transition;
END_TRANSITION
STEP S30_ProgEnd:
	S30_ProgEnd_action(N);
END_STEP
TRANSITION FROM S30_ProgEnd TO Init := TRUE;
END_TRANSITION

ACTION Start_action:
Done:=FALSE;
END_ACTION

ACTION Init_action:
(* Initialize kinematics flags*)
	AxisGroupKin_Inst.In.Cp.Settings.PlusTargetCartABC :=FALSE;
	AxisGroupKin_Inst.In.Cp.Settings.UseMasterPosition:=FALSE;

(* CP settings *)
	(* Initialize SegID *)
	AxisGroupKin_Inst.In.Cp.Segment.ID := AxisGroupKin_Inst.Out.Cp.Queue.LastMappedSegID;
	(* Initialize global point array *)
	points[1].x:=10;	points[1].y:=100;	points[1].z:=50;
	points[2].x:=10;	points[2].y:=200;	points[2].z:=100;
	points[3].x:=50;	points[3].y:=300;	points[3].z:=50;
	points[4].x:=100;	points[4].y:=350;	points[4].z:=100;
	points[5].x:=200;	points[5].y:=300;	points[5].z:=50;
	points[6].x:=300;	points[6].y:=200;	points[6].z:=100;
	points[7].x:=300;	points[7].y:=100;	points[7].z:=50;
	points[8].x:=200;	points[8].y:=50;	points[8].z:=100;
	points[9].x:=100;	points[9].y:=10;	points[9].z:=50;
	points[10].x:=50;	points[10].y:=50;	points[10].z:=100;
	(* motion parameters for CP modes *)
	AxisGroupKin_Inst.In.Cp.Segment.Translation.Velocity := 100;
	AxisGroupKin_Inst.In.Cp.Segment.Translation.Acceleration := 100;
	AxisGroupKin_Inst.In.Cp.Segment.Translation.Deceleration := 100;
	AxisGroupKin_Inst.In.Cp.Segment.Translation.Jerk := 100;
	AxisGroupKin_Inst.In.Cp.Segment.Blending.Distance := 30;
	AxisGroupKin_Inst.In.Cp.Segment.Blending.LimitationPercentage := 50;
	AxisGroupKin_Inst.In.Cp.Segment.Mode := KIN_CONTINUOUS_PATH;
	AxisGroupKin_Inst.In.Cp.Path.VelocityPercentage:=100;
	AxisGroupKin_Inst.In.Cp.Path.FidelityPercentage :=100;

(* TARGET_CART settings *)
	(* Set motion parameters for target mode*)
	AxisGroupKin_Inst.In.Target.Cart.Acceleration := CART_ACC50;
	AxisGroupKin_Inst.In.Target.Cart.Deceleration := CART_DEC50;
	AxisGroupKin_Inst.In.Target.Cart.Velocity := CART_VEL50;
	AxisGroupKin_Inst.In.Target.Cart.Jerk:=CART_Jerk100;
	AxisGroupKin_Inst.In.Target.CoordSys := KIN_KCS;
	AxisGroupKin_Inst.In.Target.Synchronization:= KIN_NO_SYNC;

	AxisGroupKin_Inst.In.General.Mode := KIN_TARGET_CART;

	i:=1;
END_ACTION

ACTION S00_TARGET_LAST_POINT_OF_ARRAY_action:
(* move to last point in array *)
AxisGroupKin_Inst.In.Target.Position[1] := points[10].x;
AxisGroupKin_Inst.In.Target.Position[2] := points[10].y;
AxisGroupKin_Inst.In.Target.Position[3] := points[10].z;
END_ACTION

ACTION S10_Fill_Queue_entry:
AxisGroupKin_Inst.In.General.Mode			:= KIN_LIN_3D;
AxisGroupKin_Inst.In.Cp.Segment.Position[1]	:= points[i].x;
AxisGroupKin_Inst.In.Cp.Segment.Position[2] 	:= points[i].y;
AxisGroupKin_Inst.In.Cp.Segment.Position[3] 	:= points[i].z;
AxisGroupKin_Inst.In.Cp.Segment.ID 		:= AxisGroupKin_Inst.In.Cp.Segment.ID + 1;

i:=i+1;
END_ACTION

ACTION S30_ProgEnd_action:
Done:=TRUE;
END_ACTION

TRANSITION Transition:
MC_KinInProximity(Threshold := 0.0,
			Position := AxisGroupKin_Inst.In.Target.Position,
			CoordSys := AxisGroupKin_Inst.In.Target.CoordSys,
			Dimension := 2#0000_0111, ActPos := AxisGroupKin_Inst.Out.General.Position)

AND
AxisGroupKin_Inst.Out.General.Standstill.ActCoordSys
END_TRANSITION

TRANSITION Transition:
(AxisGroupKin_Inst.Out.Cp.Queue.LastMappedSegID= AxisGroupKin_Inst.In.Cp.Segment.ID) AND (i >10)
END_TRANSITION

TRANSITION Transition:
AxisGroupKin_Inst.Out.Cp.Queue.LastMappedSegID = AxisGroupKin_Inst.In.Cp.Segment.ID
END_TRANSITION

TRANSITION Transition:
AxisGroupKin_Inst.Out.Cp.Path.EndReached
END_TRANSITION
END_FUNCTION_BLOCK

(* POU AxisGroupControl_Kinematics/Examples/PRG07_XYZ_USER_ST, ST *)
(*##############################################################################################################

	IMPORTANT NOTICE:
 	This example is a special and free service that demonstrates only the basic 
	approach to generating a PLC program as a non-binding sample. 
	SEW is not liable for the contents of the sample program.

	Name:			PRG_XYZ_USER_ST
	Job:			Example program
					Simple program, in which you can implement your own sample sequence.			

################################################################################################################*)
FUNCTION_BLOCK PRG07_XYZ_USER_ST
VAR_INPUT
	Enable : BOOL;
END_VAR
VAR_OUTPUT
	Active : BOOL;
	Done : BOOL;
END_VAR
VAR
	nState : INT;
	fbRtrig : R_TRIG;
END_VAR
VAR_IN_OUT
	AxisGroupKin_Inst											: ST_AxisGroupKin_Instance;
END_VAR
(* Initialisation at rising edge of VAR_INPUT Enable *)
fbRtrig(CLK:=Enable);
IF fbRtrig.Q THEN
	nState	:= 0;
	Active := TRUE;
END_IF

(* No execution, if Enable = False *)
IF NOT Enable THEN
	Done := FALSE;
	RETURN;
END_IF

CASE nState OF
0:	(*Start*)
	IF AxisGroupKin.ConfigDataAvailable THEN
		nState := 5;
	END_IF
5:	(* TARGET_CART to XYZ_USER_P1 *)
	(* Initialize Kinematic Flags*)
	AxisGroupKin_Inst.In.Cp.Settings.PlusTargetCartABC:=FALSE;
	AxisGroupKin_Inst.In.Cp.Settings.UseMasterPosition:=FALSE;

(* TARGET_CART settings *)
	(* Motion Parameters *)
	AxisGroupKin_Inst.In.Target.Cart.Velocity := CART_VEL50;
	AxisGroupKin_Inst.In.Target.Cart.Acceleration := CART_ACC50;
	AxisGroupKin_Inst.In.Target.Cart.Deceleration := CART_DEC50;
	AxisGroupKin_Inst.In.Target.Cart.Jerk:=CART_Jerk100;
	AxisGroupKin_Inst.In.Target.Synchronization:= KIN_NO_SYNC;
	(* Coordinate System *)
	AxisGroupKin_Inst.In.Target.CoordSys:=KIN_KCS;

	AxisGroupKin_Inst.In.General.Mode := KIN_TARGET_CART;

	AxisGroupKin_Inst.In.Simu3D.Ctrl.Pen_TCP_WCS := TRUE;  (* Process On *)

	AxisGroupKin_Inst.In.Target.Position := XYZ_USER_P1;
	IF (MC_KinInProximity(Threshold := 0.0,
			Position := AxisGroupKin_Inst.In.Target.Position,
			CoordSys := AxisGroupKin_Inst.In.Target.CoordSys,
			Dimension := 2#0000_0111, ActPos := AxisGroupKin_Inst.Out.General.Position)
			AND AxisGroupKin_Inst.Out.General.Standstill.ActCoordSys) THEN
		nState := 10;
	END_IF

10:	(* TARGET_CART to XYZ_USER_P2 *)
	AxisGroupKin_Inst.In.Target.Position := XYZ_USER_P2;
	IF (MC_KinInProximity(Threshold := 0.0,
			Position := AxisGroupKin_Inst.In.Target.Position,
			CoordSys := AxisGroupKin_Inst.In.Target.CoordSys,
			Dimension := 2#0000_0111, ActPos := AxisGroupKin_Inst.Out.General.Position)
			AND AxisGroupKin_Inst.Out.General.Standstill.ActCoordSys) THEN
		Done := TRUE;
		Active := FALSE;
		AxisGroupKin_Inst.In.Simu3D.Ctrl.Pen_TCP_WCS := FALSE;  (* Process Off *)
	END_IF

ELSE
;

END_CASE
END_FUNCTION_BLOCK

(* POU AxisGroupControl_Kinematics/Examples/PRG08_XYZ_USER_SFC, SFC *)
(*##############################################################################################################

	IMPORTANT NOTICE:
 	This example is a special and free service that demonstrates only the basic 
	approach to generating a PLC program as a non-binding sample. 
	SEW is not liable for the contents of the sample program.

	Name:			PRG_XYZ_USER_SFC
	Job:			Example program
					Simple program, in which you can implement your own sample sequence.				

################################################################################################################*)
FUNCTION_BLOCK PRG08_XYZ_USER_SFC
VAR_INPUT
	SFCReset:BOOL;
	(*SFCInit:BOOL;*)
	SFCPause:BOOL;

	SFCTipMode:BOOL;
	SFCTip:BOOL;
	SFCEnableLimit:BOOL;
	SFCQuitError:BOOL;

END_VAR
VAR_OUTPUT
	SFCTrans:BOOL;
	SFCError:BOOL;
	SFCErrorStep:STRING;
	SFCErrorPOU:STRING;
(*	SFCErrorAnalyzation:STRING;*)
	SFCCurrentStep:STRING;
	Done:BOOL;
END_VAR
VAR

END_VAR
VAR_IN_OUT
	AxisGroupKin_Inst											: ST_AxisGroupKin_Instance;
END_VAR
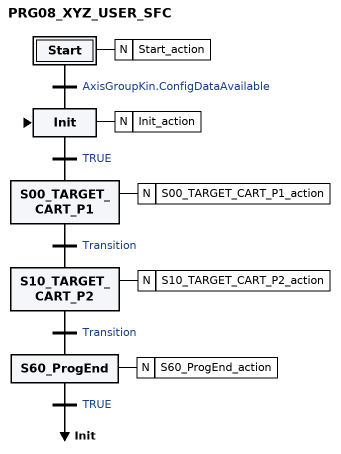
INITIAL_STEP Start:
	Start_action(N);
END_STEP
TRANSITION FROM Start TO Init := AxisGroupKin.ConfigDataAvailable;
END_TRANSITION
STEP Init:
	Init_action(N);
END_STEP
TRANSITION FROM Init TO S00_TARGET_CART_P1 := TRUE;
END_TRANSITION
STEP S00_TARGET_CART_P1:
	S00_TARGET_CART_P1_action(N);
END_STEP
TRANSITION FROM S00_TARGET_CART_P1 TO S10_TARGET_CART_P2 := Transition;
END_TRANSITION
STEP S10_TARGET_CART_P2:
	S10_TARGET_CART_P2_action(N);
END_STEP
TRANSITION FROM S10_TARGET_CART_P2 TO S60_ProgEnd := Transition;
END_TRANSITION
STEP S60_ProgEnd:
	S60_ProgEnd_action(N);
END_STEP
TRANSITION FROM S60_ProgEnd TO Init := TRUE;
END_TRANSITION

ACTION Start_action:
Done:=FALSE;
END_ACTION

ACTION Init_action:
(* Initialize Kinematic Flags*)
AxisGroupKin_Inst.In.Cp.Settings.PlusTargetCartABC:=FALSE;
AxisGroupKin_Inst.In.Cp.Settings.UseMasterPosition:=FALSE;

(* TARGET_CART settings *)
	(* Motion Parameters *)
	AxisGroupKin_Inst.In.Target.Cart.Velocity := CART_VEL50;
	AxisGroupKin_Inst.In.Target.Cart.Acceleration := CART_ACC50;
	AxisGroupKin_Inst.In.Target.Cart.Deceleration := CART_DEC50;
	AxisGroupKin_Inst.In.Target.Cart.Jerk:=CART_Jerk100;
	AxisGroupKin_Inst.In.Target.Synchronization:= KIN_NO_SYNC;
	(* Coordinate System *)
	AxisGroupKin_Inst.In.Target.CoordSys:=KIN_KCS;

AxisGroupKin_Inst.In.General.Mode := KIN_TARGET_CART;

AxisGroupKin_Inst.In.Simu3D.Ctrl.Pen_TCP_WCS := TRUE;  (* Process On *)
END_ACTION

ACTION S00_TARGET_CART_P1_action:
AxisGroupKin_Inst.In.Target.Position := XYZ_USER_P1;
END_ACTION

ACTION S10_TARGET_CART_P2_action:
AxisGroupKin_Inst.In.Target.Position := XYZ_USER_P2;
END_ACTION

ACTION S60_ProgEnd_action:
Done := TRUE;
AxisGroupKin_Inst.In.Simu3D.Ctrl.Pen_TCP_WCS := FALSE;  (* Process Off *)
END_ACTION

TRANSITION Transition:
MC_KinInProximity(Threshold := 0.0,
			Position := AxisGroupKin_Inst.In.Target.Position,
			CoordSys := AxisGroupKin_Inst.In.Target.CoordSys,
			Dimension := 2#0000_0111, ActPos := AxisGroupKin_Inst.Out.General.Position)
AND
AxisGroupKin_Inst.Out.General.Standstill.ActCoordSys
END_TRANSITION

TRANSITION Transition:
MC_KinInProximity(Threshold := 0.0,
			Position := AxisGroupKin_Inst.In.Target.Position,
			CoordSys := AxisGroupKin_Inst.In.Target.CoordSys,
			Dimension := 2#0000_0111, ActPos := AxisGroupKin_Inst.Out.General.Position)
AND
AxisGroupKin_Inst.Out.General.Standstill.ActCoordSys
END_TRANSITION
END_FUNCTION_BLOCK

(* POU PRG_Kinematics/PRG_TaskPriority_Kinematics, ST *)
PROGRAM PRG_TaskPriority_Kinematics
VAR
END_VAR
(*#######################################################################################

	PRG_TaskPriority_Kinematics

	ToDo: Call this program in the task configuration after PRG_TaskPriority();

########################################################################################*)

(* Do not remove! *)
AxisGroupControl_Priority_Kinematics();
END_PROGRAM
